(* F_GetSign indicates the sign of the input LREAL value, set to 0 is input value is 0 *)
(* 1 = +ive, -1 = -ive *)
FUNCTION F_GetSign : INT
VAR_INPUT
	fValue		: LREAL;
END_VAR
VAR
END_VAR
(*
-------------------------------------------------------------------------------------------------
Date		Version	Author	Comments
-------------------------------------------------------------------------------------------------
30/01/2015	3.00.00	PB		No change

-------------------------------------------------------------------------------------------------
05/02/10	1.00.00	PB		Initial release

-------------------------------------------------------------------------------------------------
*)

(* input value is positive *)
IF fValue > 0.0 THEN

	F_GetSign := 1;

(* input value is negative *)
ELSIF fValue < 0.0 THEN

	F_GetSign := -1;

(* input value is zero *)
ELSE

	F_GetSign := 0;
END_IF

END_FUNCTION

(* stored: Version 1.1.0.1, ProductVersion 3.1.4024.15
   POU F_GetSign: Id {0e64ecf9-9008-4df4-9153-74536ab93cc4}, SpecialFunc None *)
